FUNCTION_BLOCK FB_TestTester
VAR
END_VAR

METHOD AddTwo : DINT
VAR_INPUT
    In1 : DINT;
    In2 : DINT;
END_VAR
AddTwo := In1 + In2;
END_METHOD

PROPERTY TestBool : BOOL
GET
TestBool := TRUE;
END_GET
SET
END_SET
END_PROPERTY

PROPERTY TestLReal : LREAL
GET
TestLReal := 75.75;
END_GET
SET
END_SET
END_PROPERTY

PROPERTY TestString : STRING
GET
TestString := 'TestString';
END_GET
SET
END_SET
END_PROPERTY

END_FUNCTION_BLOCK

(* stored: Version 1.1.0.1
   POU FB_TestTester: Id {012b8ed0-2a5c-4bc2-bd74-056604d88c1c}, SpecialFunc None
   Method AddTwo: Id {2fd73b10-3d6d-4b49-8abc-ef2b87de2173}
   Property TestBool: Id {2988899c-ca12-45f9-859d-d570b073326e}
   Get Get: Id {f1d35567-8ed4-4dba-988e-94ce8ffb7c35}
   Set Set: Id {bcd3f901-a239-4e8e-a65b-26db934b60b2}
   Property TestLReal: Id {d3969fe2-4c8a-4c9e-b7f5-adf569135974}
   Get Get: Id {6dac0174-de78-4565-9f23-a2e9589d1681}
   Set Set: Id {80a86056-3cd0-4c46-b68c-e9acf38aeddd}
   Property TestString: Id {22424641-a845-4ed3-85b7-950315ad3776}
   Get Get: Id {1742c6f3-0ee6-4366-846b-5aca271d1aa5}
   Set Set: Id {2e3852b0-e84e-40d7-93eb-d5d92c41872b} *)
